(* IEC 61131-3 sources: Lasal/CPU_5344_V01/Class/MillLine, 1 file *)

(* ---- MillLine.st ---- *)
(*!
<Class
	Name               = "MillLine"
	Revision           = "0.0"
	RealtimeTask       = "false"
	CyclicTask         = "false"
	BackgroundTask     = "false"
	Sigmatek           = "false"
	OSInterface        = "false"
	HighPriority       = "false"
	Automatic          = "false"
	UpdateMode         = "Prescan"
	SharedCommandTable = "true"
	Objectsize         = "(390,360)">
	<Channels>
		<Server Name="ClassSvr" Visualized="false" Initialize="false" WriteProtected="true" Retentive="false"/>
		<Server Name="middleX" Visualized="true" Initialize="false" WriteProtected="false" Retentive="false"/>
		<Server Name="middleY" Visualized="true" Initialize="false" WriteProtected="false" Retentive="false"/>
		<Server Name="millType" Visualized="true" Initialize="false" WriteProtected="false" Retentive="false"/>
		<Server Name="radius" Visualized="true" Initialize="false" WriteProtected="false" Retentive="false"/>
		<Server Name="rnr" Visualized="true" Initialize="false" WriteProtected="false" Retentive="false"/>
		<Server Name="xGoal" Visualized="true" Initialize="false" WriteProtected="false" Retentive="false"/>
		<Server Name="yGoal" Visualized="true" Initialize="false" WriteProtected="false" Retentive="false"/>
	</Channels>
</Class>
*)
MillLine : CLASS
  //Servers:
	ClassSvr 	: SvrChCmd_DINT;
	rnr 	: SvrCh_DINT;
	millType 	: SvrCh_eMillType;
	xGoal 	: SvrCh_DINT;
	yGoal 	: SvrCh_DINT;
	radius 	: SvrCh_DINT;
	middleX 	: SvrCh_DINT;
	middleY 	: SvrCh_DINT;
  //Clients:
  //Variables:
		ptr 	: ^strMillLine;
  //Functions:

	FUNCTION GLOBAL WritePtr
		VAR_INPUT
			iPtr 	: ^strMillLine;
		END_VAR;

	FUNCTION WriteServers;

	FUNCTION VIRTUAL GLOBAL millType::Write
		VAR_INPUT
			input (EAX) 	: eMillType;
		END_VAR
		VAR_OUTPUT
			result (EAX) 	: eMillType;
		END_VAR;

	FUNCTION VIRTUAL GLOBAL xGoal::Write
		VAR_INPUT
			input (EAX) 	: DINT;
		END_VAR
		VAR_OUTPUT
			result (EAX) 	: DINT;
		END_VAR;

	FUNCTION VIRTUAL GLOBAL yGoal::Write
		VAR_INPUT
			input (EAX) 	: DINT;
		END_VAR
		VAR_OUTPUT
			result (EAX) 	: DINT;
		END_VAR;

	FUNCTION VIRTUAL GLOBAL radius::Write
		VAR_INPUT
			input (EAX) 	: DINT;
		END_VAR
		VAR_OUTPUT
			result (EAX) 	: DINT;
		END_VAR;

	FUNCTION VIRTUAL GLOBAL middleX::Write
		VAR_INPUT
			input (EAX) 	: DINT;
		END_VAR
		VAR_OUTPUT
			result (EAX) 	: DINT;
		END_VAR;

	FUNCTION VIRTUAL GLOBAL middleY::Write
		VAR_INPUT
			input (EAX) 	: DINT;
		END_VAR
		VAR_OUTPUT
			result (EAX) 	: DINT;
		END_VAR;
  //Tables:
	FUNCTION @STD
		VAR_OUTPUT
			ret_code	: CONFSTATES;
		END_VAR;
	FUNCTION GLOBAL TAB @CT_;
END_CLASS;

FUNCTION VIRTUAL GLOBAL MillLine::millType::Write
	VAR_INPUT
		input (EAX) 	: eMillType;
	END_VAR
	VAR_OUTPUT
		result (EAX) 	: eMillType;
	END_VAR

  if ptr <> NIL then
    millType := input;
    ptr^.millType := millType;
    result :=millType;
  else
    result := ACCESS_DENIED$eMillType;
  end_if;

END_FUNCTION

FUNCTION VIRTUAL GLOBAL MillLine::xGoal::Write
	VAR_INPUT
		input (EAX) 	: DINT;
	END_VAR
	VAR_OUTPUT
		result (EAX) 	: DINT;
	END_VAR

  if ptr <> NIL then
    xGoal := input;
    ptr^.xGoal := xGoal;
    result := xGoal;
  else
    result := ACCESS_DENIED;
  end_if;

END_FUNCTION

FUNCTION VIRTUAL GLOBAL MillLine::yGoal::Write
	VAR_INPUT
		input (EAX) 	: DINT;
	END_VAR
	VAR_OUTPUT
		result (EAX) 	: DINT;
	END_VAR

  if ptr <> NIL then
    yGoal := input;
    ptr^.yGoal := yGoal;
    result := yGoal;
  else
    result := ACCESS_DENIED;
  end_if;

END_FUNCTION

FUNCTION GLOBAL MillLine::WritePtr
	VAR_INPUT
		iPtr 	: ^strMillLine;
	END_VAR

  ptr := iPtr;
  WriteServers();

END_FUNCTION

FUNCTION MillLine::WriteServers

  if ptr <> NIL then
    millType := ptr^.millType;
    xGoal := ptr^.xGoal;
    yGoal := ptr^.yGoal;
    radius := ptr^.radius;
    middleX := ptr^.middleX;
    middleY := ptr^.middleY;
  end_if;

END_FUNCTION

FUNCTION VIRTUAL GLOBAL MillLine::radius::Write
	VAR_INPUT
		input (EAX) 	: DINT;
	END_VAR
	VAR_OUTPUT
		result (EAX) 	: DINT;
	END_VAR

  if ptr <> NIL then
	  radius := input;
    ptr^.radius := radius;
	  result := radius;
  else
    result := ACCESS_DENIED;
  end_if;

END_FUNCTION

FUNCTION VIRTUAL GLOBAL MillLine::middleX::Write
	VAR_INPUT
		input (EAX) 	: DINT;
	END_VAR
	VAR_OUTPUT
		result (EAX) 	: DINT;
	END_VAR

  if ptr <> NIL then
	  middleX := input;
    ptr^.middleX:=input;
	  result := middleX;
  else
    result := ACCESS_DENIED;
  end_if;

END_FUNCTION

FUNCTION VIRTUAL GLOBAL MillLine::middleY::Write
	VAR_INPUT
		input (EAX) 	: DINT;
	END_VAR
	VAR_OUTPUT
		result (EAX) 	: DINT;
	END_VAR

  if ptr <> NIL then
	  middleY := input;
    ptr^.middleY:=input;
	  result := middleY;
  else
    result := ACCESS_DENIED;
  end_if;

END_FUNCTION
